	iExecute			: I_Execute;
END_VAR
IF IsSome(_nState) THEN
	RETURN;
END_IF

IF (_iExecute := iExecute) = 0 THEN
	_nState := Err.Itf0;
	DebugMsg(THIS^, Tc2_Standard.CONCAT(__POUNAME(), ': Itf = 0!'));
	RETURN;
END_IF



IF _Runtime.iLastCyclic <> 0 THEN
	IF IsErr(_Runtime.iLastCyclic.Attach(THIS^), nOut => _nState) THEN
		DebugMsg(THIS^, Tc2_Standard.CONCAT(__POUNAME(), ': Error Inside!'));
	END_IF
ELSE
	_Runtime.iFirstCyclic := THIS^;
	_Runtime.iLastCyclic := THIS^;
	_nState := Ok;
END_IF
END_METHOD

PROPERTY Phase : INT
GET
Phase := _nPhase;
END_GET
SET
_nPhase := Phase;
END_SET
END_PROPERTY

PROPERTY INTERNAL State : Result
GET
State := _nState;
END_GET
SET
IF IsNone(_nState) THEN
	_nState := State;
END_IF
END_SET
END_PROPERTY

END_FUNCTION_BLOCK

// ---- Runtime/Runtime.TcPOU
(*
Manages the initialization and cyclic execution of registered function blocks.
*)
FUNCTION Runtime

IF _Runtime.bInit THEN
	IF _Runtime.iFirstInit <> 0 THEN
		_Runtime.iFirstInit.Init();
	END_IF
	_Runtime.bInit := FALSE;

	IF _Ec.nConstructedScopes <> 0 THEN
		DebugMsg(0, 'Close all Entity scopes!');
	END_IF
	
	IF _Debug.nErrorNumber > 0 THEN
		_Runtime.iFirstCyclic := 0;
		Tc2_System.ADSLOGSTR(Tc2_System.ADSLOG_MSGTYPE_ERROR, Tc2_Standard.CONCAT('Runtime disabled! Errors: ', UDINT_TO_STRING(_Debug.nErrorNumber)), '');
	END_IF
END_IF

IF _Runtime.iFirstCyclic <> 0 THEN
	_Runtime.iFirstCyclic.Exe();
END_IF

END_FUNCTION

// ---- State/_Buffer/_StateBuffer.TcPOU
(*
A circular buffer for storing states.  
*)
FUNCTION_BLOCK INTERNAL _StateBuffer
VAR_GENERIC CONSTANT
	STATE_CAP			: UDINT(1..16#7FFFFFFF) := 1;
END_VAR
VAR
	_iState				: ARRAY[1..STATE_CAP] OF I_StateInternal;
	_nHead				: UDINT := 1;
	_nTail				: UDINT := 1;
	_nLen				: UDINT;
END_VAR

(*
Returns the maximum capacity of the state buffer, indicating how many states it can hold.
*)
METHOD Cap : UDINT
VAR_INPUT
END_VAR
Cap := STATE_CAP;
END_METHOD

(*
Returns the current number of states stored in the buffer.
*)
METHOD Length : UDINT
VAR_INPUT
END_VAR
Length := _nLen;
END_METHOD

(*
Removes and retrieves the oldest state from the buffer.  

Returns:
- `Ok` - If a state is successfully removed.
- `None` - If the buffer is empty.
*)
METHOD Pop : Result
VAR_OUTPUT
	iState			: I_StateInternal;
END_VAR
IF _nHead = _nTail THEN
    Pop := None;
    RETURN;
END_IF

iState := _iState[_nHead];
_iState[_nHead] := 0;

_nHead := _nHead + 1;
_nLen := _nLen - 1;

IF _nHead > STATE_CAP THEN
    _nHead := 1;
END_IF

Pop := Ok;
END_METHOD

(*
Adds a new state to the buffer.  
Returns:
- `Ok` - If the state is successfully added.
- `Err.Itf0` - If the provided state interface is invalid.
- `Err.Ovf` - If the buffer is full.
*)
METHOD Push : Result
VAR_INPUT
	iState			: I_StateInternal;
END_VAR
VAR
	_nNextTail 		: UDINT;
END_VAR
IF iState = 0 THEN
	Push := Err.Itf0;
	RETURN;
END_IF

_nNextTail := _nTail + 1;

IF _nNextTail > STATE_CAP THEN
    _nNextTail := 1;
END_IF

IF _nNextTail = _nHead THEN
    Push := Err.Ovf; 
    RETURN;
END_IF

_nLen := _nLen + 1;
_iState[_nTail] := iState;
_nTail := _nNextTail;
Push := Ok;
END_METHOD

END_FUNCTION_BLOCK

// ---- State/Helpers/GetStateManager.TcPOU
(*
Searches an `I_Entity` for a `I_StateManager` component matching provided id pattern.
Result:
- Ok - Returns `I_StateManager`.
- None - Returns null.
- Err.Itf0 - Returns null, incorrect interface.
*)
FUNCTION GetStateManager : Result
VAR_INPUT
	iEntity		: I_Entity;
END_VAR
VAR_OUTPUT
	iSmgr		: I_StateManager;
END_VAR
VAR
	i			: Iter(1);
	_iComp		: I_FatComponent;
	cmp			: TagCmp;
END_VAR

IF iEntity = 0 THEN
	GetStateManager := Err.Itf0;
	RETURN;
END_IF

WHILE IsOk(iEntity.Get(i.Next(), iComp => _iComp)) DO
	IF IsOk(ICompToIStateMgr(_iComp.Raw, iDest => iSmgr)) THEN
		GetStateManager := Ok;
		RETURN;
	END_IF
END_WHILE

END_FUNCTION

// ---- State/Manager/ICompToIStateMgr.TcPOU
(*
Casts I_Component as I_StateManager.
Returns:
- Ok - Success,
- Err.InvRef - Invalid reference,
- Err.Itf0 - Invalid interface,
- Err.NoMatch - Cast failed
*)
FUNCTION ICompToIStateMgr : Result
VAR_INPUT
	iIn		: I_Component;
	iOut	: REFERENCE TO I_StateManager;
END_VAR

IF NOT __ISVALIDREF(iOut) THEN
	ICompToIStateMgr := Err.InvRef;
	RETURN;
END_IF

IF iIn = 0 THEN
	ICompToIStateMgr := Err.Itf0;
	RETURN;
END_IF

IF __QUERYINTERFACE(iIn, iOut) THEN
	ICompToIStateMgr := Ok;
ELSE
	ICompToIStateMgr := Err.NoMatch;
END_IF

END_FUNCTION

// ---- State/Helpers/GetState.TcPOU
(*
Searches an `I_Entity` for a `I_State` component matching provided id pattern.
Result:
- Ok - Returns `I_State`.
- Err.NotFound - Returns null.
- Err.InvRef - Returns null.
- Err.Itf0 - Returns null, incorrect interface.
*)
FUNCTION GetState : Result
VAR_INPUT
	iEntity		: I_Entity;
	sTagId		: Str;
	iOut		: REFERENCE TO I_State;
END_VAR
VAR
	i			: Iter(1);
	_iComp		: I_FatComponent;
	cmp			: TagCmp;
END_VAR

IF iEntity = 0 THEN
	GetState := Err.Itf0;
	RETURN;
END_IF

IF NOT __ISVALIDREF(iOut) THEN
	GetState := Err.InvRef;
	RETURN;
END_IF

WHILE IsOk(iEntity.Get(i.Next(), _iComp)) DO
	IF IsOk(ICompToIState(_iComp.Raw, iOut)) THEN
		IF cmp.Set(iOut.Tag).MatchWcdId(sTagId).IsTrue() THEN
			GetState := Ok;
			RETURN;
		ELSE
			iOut := 0;
		END_IF
	END_IF
END_WHILE

GetState := Err.NotFound;

END_FUNCTION

// ---- State/State/ICompToIState.TcPOU
(*
Casts I_Component to I_State
*)
FUNCTION ICompToIState : Result
VAR_INPUT
	iSource	: I_Component;
END_VAR
VAR_OUTPUT
	iDest	: I_State;
END_VAR

IF iSource = 0 THEN
	ICompToIState := Err.Itf0;
	RETURN;
END_IF

IF __QUERYINTERFACE(iSource, iDest) THEN
	ICompToIState := Ok;
ELSE
	iDest := 0;
	ICompToIState := Err.NoMatch;
END_IF

END_FUNCTION

// ---- State/_Machine/_StateMachine.TcPOU
FUNCTION_BLOCK INTERNAL _StateMachine IMPLEMENTS I_Execute
VAR
	_exe					: Execute(THIS^);
	_iCurrentState			: I_StateInternal;
END_VAR

(*
Changes the current state to a new state.  

Returns:
- `Ok` - If the state transition is successful.
- `Err.Itf0` - If the new state interface is invalid.
- `None` - If the transition cannot be completed due to state conditions.
*)
METHOD Change : Result
VAR_INPUT
	iNewState	: I_StateInternal;
END_VAR
VAR_OUTPUT
	iOldState	: I_StateInternal;
END_VAR
IF iNewState = 0 THEN
	Change := Err.Itf0;
	RETURN;
END_IF

IF iNewState = _iCurrentState THEN
	Change := None;
	RETURN;
END_IF

IF NOT iNewState._CanActivate() THEN
	Change := None;
	RETURN;
END_IF

IF _iCurrentState <> 0 AND_THEN NOT _iCurrentState._CanDeactivate() THEN
	Change := None;
	RETURN;
END_IF

IF _iCurrentState <> 0 THEN
	_iCurrentState._OnExit();
END_IF

iNewState._OnEntry();
iOldState := _iCurrentState;
_iCurrentState := iNewState;
Change := Ok;
END_METHOD

METHOD Execute
VAR_INPUT
	nPhase: INT := 0;
END_VAR
IF _iCurrentState <> 0 THEN
	_iCurrentState._OnExecute();
END_IF
END_METHOD

(*
Provides access to the current state, enabling inspection or external interaction with the state.
*)
PROPERTY State : I_State
GET
State := _iCurrentState._AsIState;
END_GET
END_PROPERTY

END_FUNCTION_BLOCK

// ---- State/Manager/StateManager.TcPOU
(*
Manages the lifecycle and transitions of states within an entity.  
Supports queuing state change requests, triggering state transitions, and broadcasting state change events.  
Adds a `_stateChangeEvent` Signal to the owning `I_Entity` during initialization, enabling external components to listen for state changes.
*)
FUNCTION_BLOCK FINAL StateManager IMPLEMENTS I_Execute, I_StateManager, I_Debug

VAR
	_comp				: Component(THIS^);

	_exe				: Execute(THIS^);
	_sm					: _StateMachine;
	_buffer				: _StateBuffer;
	
	_stateChangeEvent	: Signal;
	
	_iPretender			: I_State;
	_iCurrent			: I_State;
	_iPrevious 			: I_State;
	
	
END_VAR

(*
Retrieves the currently active state managed by the state manager.
*)
PROPERTY Current : I_State
GET
Current := _iCurrent;
END_GET
END_PROPERTY

// DO NOT CALL MANUALLY
{attribute 'hide'}
METHOD Execute
VAR
	_iNewState		: I_StateInternal;
	_iOldState		: I_StateInternal;
END_VAR
IF IsOk(_buffer.Pop(iState => _iNewState)) THEN
	_iPretender := _iNewState._AsIState;
	IF IsOk(_sm.Change(_iNewState, iOldState => _iOldState)) THEN
		_stateChangeEvent.Emit(_iNewState._AsIState.Tag);
		
		_iCurrent		:= _iNewState._AsIState;
		IF _iOldState <> 0 THEN
			_iPrevious		:= _iOldState._AsIState;
		END_IF
		
	END_IF
	
	_iPretender		:= 0;
END_IF
END_METHOD

(*
Returns the entity that owns this state.
*)
PROPERTY Owner : I_Entity
GET
Owner := _comp.Entity;
END_GET
END_PROPERTY

(*
Retrieves the state that is queued to become active next, but has not yet transitioned.
*)
PROPERTY Pretender : I_State
GET
Pretender := _iPretender;
END_GET
END_PROPERTY

(*
Retrieves the last active state prior to the current one.
*)
PROPERTY Previous : I_State
GET
Previous := _iPrevious;
END_GET
END_PROPERTY

(*
Allows initializing an external interface variable with an interface pointer to this instance within declaration block.
Example:
iSMgr: I_StateManager;
smgr: StateManager := (Proxy := iSMgr);
Result: iSMgr <> 0 
*)
PROPERTY Proxy : REFERENCE TO I_StateManager
SET
Proxy := THIS^;
END_SET
END_PROPERTY

(*
Queues a request to transition to a specified state.  
Returns:
- `Ok` - If the state change request is successfully queued.
- `Err.Itf0` - If the provided state interface is invalid.
- `Err.NoMatch` - If the state does not belong to the same entity.
- `Err.IncArg` - If the state is already in the queue.
*)
METHOD Request : Result
VAR_INPUT
	iState			: I_State;
END_VAR
VAR
	iStateInternal	: I_StateInternal;
END_VAR
IF iState = 0 THEN
	Request := Err.Itf0;
	RETURN;
END_IF

IF iState.Owner <> _comp.Entity THEN
	Request := Err.NoMatch;
	RETURN;
END_IF

Request := _buffer.Push(iState._AsIStateInternal);
END_METHOD

END_FUNCTION_BLOCK

// ---- Strings/Strb/Strb.TcPOU
// A string builder utility that allows for manipulation of a string up to 255 characters. It implements the I_Strb interface that allows for method chaining.
FUNCTION_BLOCK FINAL Strb IMPLEMENTS I_Strb
VAR
	_sString	: Str;
	_nLength	: INT;
END_VAR

PROPERTY PRIVATE _this : I_Strb
GET
VAR
	_iThis : I_Strb := THIS^;
END_VAR
_this := _iThis;
END_GET
END_PROPERTY

// Appends the specified string to the current string.
// Truncates if the total length exceeds 255 characters.
METHOD Append : I_Strb
VAR_INPUT
    sToAdd : Str; // String to append
END_VAR

VAR
	_nNewLength	: INT;
END_VAR
Append := _this;

IF sToAdd = '' THEN
	RETURN;
END_IF

_nNewLength := Tc2_Standard.LEN(sToAdd) + _nLength;
IF _nNewLength > 255 THEN
	_nNewLength := 255;
END_IF

_sString := Tc2_Standard.CONCAT(_sString, sToAdd);
_nLength := _nNewLength;
END_METHOD

// Finds the first occurrence of a substring after the specified position.
// Outputs the start and end positions of the found substring.
METHOD FindFirstAfter : I_Strb
VAR_INPUT
    sToFind : Str;      // Substring to find
    nPosition : INT := 1; // Starting position for search
END_VAR
VAR_OUTPUT
    nStart : INT;       // Start position of the found substring
    nEnd : INT;         // End position of the found substring
END_VAR

VAR
	_sTemp			: Str;
	_nOffset		: INT;
END_VAR
FindFirstAfter := _this;

IF sToFind = '' THEN
	RETURN;
END_IF

IF nPosition = 0 THEN
	RETURN;
END_IF

_sTemp := Tc2_Standard.MID(_sString, _nLength, nPosition);
IF (_nOffset := Tc2_Standard.FIND(_sTemp, sToFind)) <> 0 THEN
	nStart := nPosition + _nOffset - 1;
	nEnd := nPosition + _nOffset - 2 + Tc2_Standard.LEN(sToFind);
END_IF
END_METHOD

// Finds the last occurrence of a substring before the specified position.
// Outputs the start and end positions of the found substring.
METHOD FindLastBefore : I_Strb
VAR_INPUT
    sToFind : Str;        // Substring to find
    nPosition : INT := 256; // Starting position for reverse search
END_VAR
VAR_OUTPUT
    nStart : INT;         // Start position of the found substring
    nEnd : INT;           // End position of the found substring
END_VAR
VAR
	_sTemp			: Str;
	_nFindLength	: INT := Tc2_Standard.LEN(sToFind);
	_nOffset		: INT;
END_VAR
FindLastBefore := _this;

IF sToFind = '' THEN
	RETURN;
END_IF

IF nPosition = 0 THEN
	RETURN;
END_IF

IF nPosition = 256 THEN
	nPosition := _nLength;
END_IF

REPEAT
	_sTemp := Tc2_Standard.MID(_sString, _nFindLength, nPosition);
	IF _sTemp = sToFind THEN
		nStart 	:= nPosition;
		nEnd	:= nPosition + _nFindLength - 1;
		RETURN;
	END_IF
UNTIL
	(nPosition := nPosition - 1) <= 0
END_REPEAT
END_METHOD

// Checks if the specified substring exists after the given position.
METHOD HasAfter : BOOL
VAR_INPUT
    sToFind : Str;      // Substring to search for
    nPosition : INT := 0; // Starting position for search
END_VAR
VAR_OUTPUT
    nStart : INT;       // Start position of the found substring
    nEnd : INT;         // End position of the found substring
END_VAR
FindFirstAfter(sToFind, nPosition, nStart => nStart, nEnd => nEnd);
HasAfter := nStart > 0;
END_METHOD

// Checks if the specified substring exists before the given position.
METHOD HasBefore : BOOL
VAR_INPUT
    sToFind : Str;        // Substring to search for
    nPosition : INT := 256; // Ending position for reverse search
END_VAR
VAR_OUTPUT
    nStart : INT;         // Start position of the found substring
    nEnd : INT;           // End position of the found substring
END_VAR
IF nPosition = 256 THEN
	nPosition := Tc2_Standard.LEN(_sString);
END_IF

FindLastBefore(sToFind, nPosition, nStart => nStart, nEnd => nEnd);
HasBefore := nStart > 0;
END_METHOD

// Inserts a specified substring at a given position.
// Truncates if the total length exceeds 255 characters.
METHOD Inject : I_Strb
VAR_INPUT
    nPosition : INT;    // Position to inject the string
    sToInject : Str;    // String to inject
END_VAR
VAR
	_nNewLength	: INT;
END_VAR
Inject := _this;

IF sToInject = '' THEN
	RETURN;
END_IF

IF nPosition = 0 THEN
	RETURN;
END_IF

IF nPosition > _nLength THEN
	RETURN;
END_IF

_nNewLength := Tc2_Standard.LEN(sToInject) + _nLength;
IF _nNewLength > 255 THEN
	_nNewLength := 255;
END_IF

_sString := Tc2_Standard.INSERT(_sString, sToInject, nPosition);
_nLength := _nNewLength;
END_METHOD

// Checks if the current string is empty.
METHOD IsEmpty : BOOL
VAR_INPUT
END_VAR
IsEmpty := _nLength = 0;
END_METHOD

// Returns the current length of the string.
// The length of the string is stored as a separate variable (_nLength) 
// and reflects the actual length of the content.
// Unlike Tc2_Standard.LEN(), which counts up to the first null character, 
// this method directly returns the stored length.
METHOD Length : INT
VAR_INPUT
END_VAR
Length := _nLength;
END_METHOD

// Prepends the specified string to the current string.
// Truncates if the total length exceeds 255 characters.
METHOD Prepend : I_Strb
VAR_INPUT
    sToAdd : Str; // String to prepend
END_VAR
VAR
	_nNewLength	: INT;
END_VAR
Prepend := _this;

IF sToAdd = '' THEN
	RETURN;
END_IF

_nNewLength := Tc2_Standard.LEN(sToAdd) + _nLength;
IF _nNewLength > 255 THEN
	_nNewLength := 255;
END_IF

_sString := Tc2_Standard.CONCAT(sToAdd, _sString);
_nLength := _nNewLength;
END_METHOD

// Returns the current string value.
METHOD Read : Str
VAR_INPUT
END_VAR
Read := _sString;
END_METHOD

// Removes a substring of specified length starting at a given position.
METHOD Remove : I_Strb
VAR_INPUT
    nLength : INT;    // Length of the substring to remove
    nPosition : INT;  // Starting position of the substring to remove
END_VAR

VAR
	_nPosition	: INT;
END_VAR
Remove := _this;

IF nPosition = 0 THEN
	RETURN;
END_IF

IF nPosition > _nLength THEN
	RETURN;
END_IF

IF nLength = 0 THEN
	RETURN;
END_IF

IF nLength + nPosition > _nLength THEN
	nLength := _nLength - nPosition + 1;
END_IF

_sString := Tc2_Standard.DELETE(_sString, nLength, nPosition);
_nLength := _nLength - nLength;
END_METHOD

// Sets the current string to a new value.
METHOD Set : I_Strb
VAR_INPUT
    sLiteral : Str; // New string value
END_VAR
Set 		:= _this;

_sString 	:= sLiteral;
_nLength	:= Tc2_Standard.LEN(sLiteral);
END_METHOD

// Extracts a substring starting from a given position with a specified length.
METHOD Slice : I_Strb
VAR_INPUT
    nPosition : INT; // Starting position of the slice
    nLength : INT;   // Length of the slice
END_VAR
VAR_OUTPUT
    sSlice : Strb;   // The sliced string
END_VAR
Slice := _this;

IF nPosition = 0 THEN
	RETURN;
END_IF

IF nLength = 0 THEN
	RETURN;
END_IF

sSlice.Set(Tc2_Standard.MID(_sString, nLength, nPosition));
END_METHOD

// Splits the string into two parts at the specified position.
METHOD Split : I_Strb
VAR_INPUT
    nPosition : INT; // Position to split the string
END_VAR
VAR_OUTPUT
    sLeft : Strb;    // Left part of the split
    sRight : Strb;   // Right part of the split
END_VAR
Split := _this;

IF nPosition = 0 THEN
	RETURN;
END_IF

sLeft.Set(Tc2_Standard.LEFT(_sString, nPosition));
sRight.Set(Tc2_Standard.RIGHT(_sString, _nLength - nPosition));
END_METHOD

END_FUNCTION_BLOCK

// ---- Strings/Strf/Strf.TcPOU
// The Strf provides utilities for string formatting.
PROGRAM Strf

// Adds left and/or right padding to a string with a specified fill character.
// Returns the padded string.
METHOD Padding : Str
VAR_INPUT
    sValue       : Str;  // The original string
    nLeftPadding : USINT := 0; // Number of padding characters to add to the left
    nRightPadding: USINT := 0; // Number of padding characters to add to the right
    sFillChar    : Ch := ' ';  // Character used for padding
END_VAR
VAR
	_sBase					: Strb;
	_sLeft					: Strb;
	_sRight					: Strb;
END_VAR
_sBase.Set(sValue);
IF nRightPadding = 0 THEN
	WHILE _sBase.Length() < nLeftPadding DO
		_sBase.Prepend(sFillChar);
	END_WHILE
ELSIF nLeftPadding = 0 THEN
	WHILE _sBase.Length() < nRightPadding DO
		_sBase.Append(sFillChar);
	END_WHILE
ELSE
	_sBase.Split(_sBase.Length()/2, sLeft => _sLeft, sRight => _sRight);
	WHILE _sLeft.Length() < nLeftPadding DO
		_sLeft.Prepend(sFillChar);
	END_WHILE
	WHILE _sRight.Length() < nRightPadding DO
		_sRight.Append(sFillChar);
	END_WHILE
	
	_sLeft.Append(_sRight.Read());
	_sBase.Set(_sLeft.Read());
END_IF

Padding := _sBase.Read();
END_METHOD

// Converts a TIME value to a human-readable string with specified minimum and maximum units.
// Returns the formatted time string.
METHOD SimpleTime : Str
VAR_INPUT
    tValue   : TIME;  // Time value to convert
    sMinUnit : Str := 'MS'; // Minimum unit (e.g., MS, S, M, H, D)
    sMaxUnit : Str := 'S';  // Maximum unit (e.g., MS, S, M, H, D)
END_VAR
VAR
	_nMinUnit	: USINT;
	_nMaxUnit	: USINT;
	_sValues	: ARRAY[1..5] OF Strb;
	_nValues	: ARRAY[1..5] OF UINT;
	_sUnits   	: ARRAY[1..5] OF STRING := ['MS', 'S', 'M', 'H', 'D'];
	_stTime		: Tc2_Utilities.OTSTRUCT;
	_i			: USINT;
	_strb		: Strb;
END_VAR
FOR _i := 1 TO 5 DO
	IF _sUnits[_i] = sMinUnit THEN
		_nMinUnit := _i;
	END_IF
	IF _sUnits[_i] = sMaxUnit THEN
		_nMaxUnit := _i;
	END_IF
END_FOR

IF _nMaxUnit = 0 THEN
	RETURN;
END_IF

IF _nMinUnit = 0 THEN
	RETURN;
END_IF

IF _nMinUnit > _nMaxUnit THEN
	RETURN;
END_IF

_stTime := Tc2_Utilities.TIME_TO_OTSTRUCT(tValue);
_stTime.wDay := _stTime.wWeek * 7 + _stTime.wDay;

_nValues[1] := WORD_TO_UINT(_stTime.wMilliseconds);
_nValues[2] := WORD_TO_UINT(_stTime.wSecond);
_nValues[3] := WORD_TO_UINT(_stTime.wMinute);
_nValues[4] := WORD_TO_UINT(_stTime.wHour);
_nValues[5] := WORD_TO_UINT(_stTime.wDay);

_sValues[1].Set(Strf.Padding(UINT_TO_STRING(_nValues[1]), 3, 0, '0')).Append('ms');
_sValues[2].Set(Strf.Padding(UINT_TO_STRING(_nValues[2]), 2, 0, '0')).Append('s');
_sValues[3].Set(Strf.Padding(UINT_TO_STRING(_nValues[3]), 2, 0, '0')).Append('m');
_sValues[4].Set(Strf.Padding(UINT_TO_STRING(_nValues[4]), 2, 0, '0')).Append('h');
_sValues[5].Set(Strf.Padding(UINT_TO_STRING(_nValues[5]), 3, 0, '0')).Append('d');

IF _nMaxUnit < 5 THEN
    FOR _i := 5 TO _nMaxUnit + 1 BY -1 DO
        IF _nValues[_i] <> 0 THEN
            _strb.Append(_sValues[_i].Read()).Append(' ');
        END_IF
    END_FOR
END_IF

FOR _i := _nMaxUnit TO _nMinUnit BY -1 DO
    _strb.Append(_sValues[_i].Read()).Append(' ');
END_FOR

SimpleTime := _strb.Read();
END_METHOD

END_PROGRAM

// ---- Tags/Casts/IArgToITag.TcPOU
(*
Casts I_Arg to I_Tag
*)
FUNCTION IArgToITag : Result
VAR_INPUT
	iSource		: I_Arg;
END_VAR
VAR_OUTPUT
	iDest		: I_Tag;
END_VAR

IF iSource = 0 THEN
	IArgToITag := Err.Itf0;
	RETURN;
END_IF

IF __QUERYINTERFACE(iSource, iDest) THEN
	IArgToITag := Ok;
ELSE
	iDest := 0;
	IArgToITag := Err.NoMatch;
END_IF

END_FUNCTION

// ---- Tags/Casts/ICompToITag.TcPOU
(*
Casts I_Component as I_Tag.
Returns:
- Ok - Success,
- Err.InvRef - Invalid reference,
- Err.Itf0 - Invalid interface,
- Err.NoMatch - Cast failed
*)
FUNCTION ICompToITag : Result
VAR_INPUT
	iIn		: I_Component;
	iOut	: REFERENCE TO I_Tag;
END_VAR

IF NOT __ISVALIDREF(iOut) THEN
	ICompToITag := Err.InvRef;
	RETURN;
END_IF

IF iIn = 0 THEN
	ICompToITag := Err.Itf0;
	RETURN;
END_IF

IF __QUERYINTERFACE(iIn, iOut) THEN
	ICompToITag := Ok;
ELSE
	ICompToITag := Err.NoMatch;
END_IF

END_FUNCTION

// ---- Tags/Casts/ICompToITagged.TcPOU
(*
Casts I_Component as I_Tagged.
Returns:
- Ok - Success,
- Err.InvRef - Invalid reference,
- Err.Itf0 - Invalid interface,
- Err.NoMatch - Cast failed
*)
FUNCTION ICompToITagged : Result
VAR_INPUT
	iIn		: I_Component;
	iOut	: REFERENCE TO I_Tagged;
END_VAR

IF NOT __ISVALIDREF(iOut) THEN
	ICompToITagged := Err.InvRef;
	RETURN;
END_IF

IF iIn = 0 THEN
	ICompToITagged := Err.Itf0;
	RETURN;
END_IF

IF __QUERYINTERFACE(iIn, iOut) THEN
	ICompToITagged := Ok;
ELSE
	ICompToITagged := Err.NoMatch;
END_IF

END_FUNCTION

// ---- Tags/Helpers/GetTag.TcPOU
(*
Searches an `I_Entity` for a `I_Tag` component matching provided id pattern.
Result:
- Ok - Returns iTag.
- Err.NotFound - Returns null.
- Err.InvRef - Provided reference is invalid.
- Err.Itf0 - Returns null, incorrect interface.
*)
FUNCTION GetTag : Result
VAR_INPUT
	iEntity		: I_Entity;
	sIdPattern	: Str;
	iOut		: REFERENCE TO I_Tag;
END_VAR
VAR
	i			: Iter(1);
	_iComp		: I_FatComponent;
	cmp			: TagCmp;
END_VAR

IF iEntity = 0 THEN
	GetTag := Err.Itf0;
	RETURN;
END_IF

IF NOT __ISVALIDREF(iOut) THEN
	GetTag := Err.InvRef;
	RETURN;
END_IF

WHILE IsOk(iEntity.Get(i.Next(), _iComp)) DO
	IF IsOk(ICompToITag(_iComp.Raw, iOut)) THEN
		IF cmp.Set(iOut).MatchWcdId(sIdPattern).IsTrue() THEN
			GetTag := Ok;
			RETURN;
		ELSE
			iOut := 0;
		END_IF
	END_IF
END_WHILE

GetTag := Err.NotFound;

END_FUNCTION

// ---- Tags/Helpers/HasTagOption.TcPOU
(*
Searches an `I_Entity` for a `I_Tag` component with provided `Option` value.
Result:
- Ok
- Err.NotFound - Returns null.
- Err.Itf0 - Returns null, incorrect interface.
*)
FUNCTION HasTagOption : Result
VAR_INPUT
	iEntity		: I_Entity;
	sOption		: Str;
END_VAR
VAR
	i			: Iter(1);
	_iComp		: I_FatComponent;
	_iTag		: I_Tag;
END_VAR

IF iEntity = 0 THEN
	HasTagOption := Err.Itf0;
	RETURN;
END_IF

WHILE IsOk(iEntity.Get(i.Next(), _iComp)) DO
	IF IsOk(ICompToITag(_iComp.Raw, _iTag)) THEN
		IF _iTag.Option = sOption THEN
			HasTagOption := Ok;
			RETURN;
		END_IF
	END_IF
END_WHILE

HasTagOption := Err.NotFound;

END_FUNCTION

// ---- Tags/Helpers/HasTag.TcPOU
(*
Searches an `I_Entity` for a `I_Tag` component matching provided id pattern.
Result:
- Ok
- Err.NotFound - Returns null.
- Err.Itf0 - Returns null, incorrect interface.
*)
FUNCTION HasTag : Result
VAR_INPUT
	iEntity		: I_Entity;
	sIdPattern	: Str;
END_VAR
VAR
	i			: Iter(1);
	_iComp		: I_FatComponent;
	_iTag		: I_Tag;
	cmp			: TagCmp;
END_VAR

IF iEntity = 0 THEN
	HasTag := Err.Itf0;
	RETURN;
END_IF

WHILE IsOk(iEntity.Get(i.Next(), _iComp)) DO
	IF IsOk(ICompToITag(_iComp.Raw, _iTag)) THEN
		IF cmp.Set(_iTag).MatchWcdId(sIdPattern).IsTrue THEN
			HasTag := Ok;
			RETURN;
		END_IF
	END_IF
END_WHILE

HasTag := Err.NotFound;

END_FUNCTION

// ---- Tags/Helpers/MatchPath.TcPOU
(*
Returns whether the symbol's path matches the provided pattern.
Allows wildcards in form of "*" that can cover multiple segments.
Example pattern: *.functionBlock.*.bBool
*)
FUNCTION MatchPath : Result
VAR_INPUT
    sAddress : Str;  /// The symbol's path to evaluate
    sPattern : Str;  /// The pattern to match against
END_VAR
VAR
	pttPath				: TagPath;
	pttSeg				: Str;
	pttPeek				: Str;
	addPath				: TagPath;
	addSeg				: Str;
	bMatch				: BOOL;
END_VAR

// Init
IF IsErr(addPath.Set(sAddress)) THEN
	RETURN;
END_IF
IF IsErr(pttPath.Set(sPattern)) THEN
	RETURN;
END_IF

// Advance to the next segment
WHILE IsOk(pttPath.Next(sSeg => pttSeg)) DO	
	bMatch := FALSE;
	// If the current segment is a wildcard, then peek to the next segment
	IF pttSeg = '*' THEN
		IF IsOk(pttPath.Peek(sSeg => pttPeek)) THEN
			IF pttPeek = '*' THEN
				CONTINUE; // Skip redundant wildcard if *.*.
			END_IF
		ELSE
			MatchPath := Ok;
			RETURN; // No more segments in the pattern, so it's a match as everything so far matched(.*)
		END_IF

	// If current segment is not a wildcard reset the peek.
	ELSIF pttSeg <> '*' THEN
		pttPeek := '';
	END_IF
	
	// Get the next segment of the address path
	WHILE IsOk(addPath.Next(sSeg => addSeg)) DO
		IF pttPeek <> '' THEN
			IF pttPeek = addSeg THEN
				bMatch := TRUE;
				pttPath.Next(); // Consume get next pattern segment
				EXIT;
			ELSE
				CONTINUE; // Get next address
			END_IF
		ELSIF pttSeg = addSeg THEN
			bMatch := TRUE;
			EXIT; // Consume get next pattern segment
		ELSE
			RETURN; // No match - return
		END_IF
	END_WHILE

	IF NOT bMatch THEN
		RETURN;
	END_IF

END_WHILE

IF IsOk(addPath.Peek()) THEN
	RETURN;
END_IF

MatchPath := Ok;

END_FUNCTION
